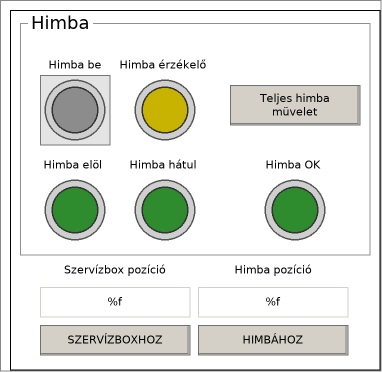
VISUALIZATION Himba  // 382x372
    Rectangle (10,10 370x360)
    GroupBox (20,15 350x240), "Himba"
        PushSwitch (20,60 70x70), variable: HIMBA.bHimba, behaviour: TOGGLE, style: Switch-PushSwitch-Gray
        Label (20,40 70x20), "Himba be"
        Group (0,140 106x90)
            Label (0,0 106x20), "Himba elöl"
            Lamp1 (20,20 70x70), variable: HIMBA.bHimba_elol, style: Lamp-Lamp1-Green
        Group (90,40 106x90)
            Lamp1 (20,20 70x70), variable: HIMBA.bHimba_szenzor, invisible if: GVL.bPtKameraTrigger OR GVL.bPtKameraHegesztesOK, style: Lamp-Lamp1-Yellow
            Label (0,0 106x20), "Himba érzékelő"
        Group (90,140 106x90)
            Lamp1 (20,20 70x70), variable: HIMBA.bHimba_hatul, style: Lamp-Lamp1-Green
            Label (0,0 106x20), "Himba hátul"
        Group (220,140 106x90)
            Lamp1 (20,20 70x70), variable: GVL.bHimbaOK, style: Lamp-Lamp1-Green
            Label (0,0 106x20), "Himba OK"
        Button (210,70 130x40), "Teljes himba müvelet", input disabled if: HIMBA.bHimba_elol=HIMBA.bHimba_hatul
            OnMouseUp: execute { HIMBA.s_InCommand:='START'; }
    Textfield (40,287 150x30), "%f", text variable: GVL.lrPtSzervizbox
    Button (40,325 150x30), "SZERVÍZBOXHOZ"
        OnMouseUp: execute { PISTITENGELY.lrPistiPosition:=GVL.lrPtSzervizbox; PISTITENGELY.sPistiAxisCommand:='MOVE'; }
    Label (40,260 150x20), "Szervízbox pozíció"
    Textfield (198,287 150x30), "%f", text variable: GVL.lrPtKameraPosition
        OnMouseClick: write the text variable via VisuDialogs.Numpad, min -10000, max -1
    Button (198,325 150x30), "HIMBÁHOZ"
        OnMouseUp: execute { PISTITENGELY.lrPistiPosition:=GVL.lrHegesztoPosition6; PISTITENGELY.sPistiAxisCommand:='MOVE'; }
    Label (198,260 150x20), "Himba pozíció"
END_VISUALIZATION

(* stored: Version 1.1.0.1, ProductVersion 3.1.4024.11
   Visu Himba: Id {73d4033e-8d5b-4993-8316-72856904c939} *)
